Fanuc KAREL source: kt00614.KL

-- PROVISIONAL review KL for V770-1; original PC SHA256 9ab1ac22b095cd8de1ef48ccaea931d284292e8ef3a96d3b23c97661c16bcc19
-- Incomplete behavior may be omitted. Consult companion uncertainty JSON. Do not deploy.
PROGRAM KT00614
%NOLOCKGROUP
VAR
  R1 : REAL
  R2 : REAL
  OUT : REAL
BEGIN
  -- UNRESOLVED_PC offsets 5-16; opcodes 2E,23
  -- UNRESOLVED_PC offsets 21-32; opcodes 2E,23
  -- UNRESOLVED_PC offsets 37-48; opcodes 2E,23
  -- UNRESOLVED_PC offsets 53-64; opcodes 2E,23
  -- UNRESOLVED_PC offsets 69-82; opcodes 21,68,23
  -- UNRESOLVED_PC offsets 87-91; opcodes 7F
END KT00614
